Fanuc KAREL source: port_LAI.kl

PROGRAM TP
%NOLOCKGROUP
VAR
 x: INTEGER
BEGIN
 x = LAI[3]
END TP
